   Drum."Step".Ons_StrobeWorkDone := FALSE;
   Drum."Step".Ons_StrobeRejectByCycleInterruption := FALSE;
   Drum."Step".StrobeWorkDone := FALSE;
   Drum."Step".StrobeRejectByCycleInterruption := FALSE;
   Drum."Step".ScSeqOk := FALSE;
   Drum."Step".SeqActive := FALSE;
   Drum.Drive.AlmOk := FALSE;
   Drum.Drive.AlmEmerg := FALSE;
   Drum.Drive.AlmNode := FALSE;
   Drum.Drive.InitPosDrive := FALSE;
   Drum.Drive.InitPosDrivePLS := FALSE;
   Drum.Drive.GearingON := FALSE;
   Drum.Drive.CamHook := FALSE;
   Drum.Drive.CamStoppingPhase := FALSE;
   Drum.Drive.RepositioningRequest := FALSE;
   Drum.Drive.CamRequestResult := FALSE;
   Drum.Drive.CamRequestError := FALSE;
   Drum.Drive.CamRequestOk := TRUE;
   Drum.Drive.CalibDisAxisReq := FALSE;
   Drum.Drive.CalibReq := FALSE;
   Drum.Drive.CalibProcess := FALSE;
   Drum.Drive.HwOvertravelDisReq := FALSE;
   Drum.Drive.HwOvertravelEnReq := FALSE;
   Drum.Drive.AuxCamRequest := FALSE;
   Drum.Drive.TorquePeakEna := FALSE;
   Drum.Drive.Cmd_Repos := FALSE;
   Drum.Drive.Ons_CamRequest := FALSE;
   Drum.Drive.AuxCmdPosition := 0;
   Drum.Drive.Unwind := 90.0;
   Drum.Drive.MaxDev := 30.0;
   Drum.Drive.ReposSpeed := 10.0;
   Drum.Drive.CalcSlaveDifferenceABS := 0.0;
   Drum.Drive.CalcModPosition := 0.0;
   Drum.Drive.CalcSlaveDifference := 0.0;
   Drum.Drive.CalcMinDeltaPos := 0.0;
   Drum.Drive.CalcMaxDeltaPos := 0.0;
   Drum.Drive.CalcHalfPosUnwind := 0.0;
   Drum.Drive.Man.Cmd_PosJog := FALSE;
   Drum.Drive.Man.Cmd_NegJog := FALSE;
   Drum.Drive.Man.Cmd_Step := FALSE;
   Drum.Drive.Man.Cmd_Forward := FALSE;
   Drum.Drive.Man.Cmd_Backward := FALSE;
   Drum.Drive.Man.Cmd_Up := FALSE;
   Drum.Drive.Man.Cmd_Down := FALSE;
   Drum.Drive.Man.Cmd_Intermediate := FALSE;
   Drum.Drive.Man.Cmd_Open := FALSE;
   Drum.Drive.Man.Cmd_Close := FALSE;
   Drum.Drive.Man.Cmd_PreOpen := FALSE;
   Drum.Drive.Man.Cmd_Maintenance := FALSE;
   Drum.Drive.Man.Cmd_OperatorSide := FALSE;
   Drum.Drive.Man.Cmd_NotOperatorSide := FALSE;
   Drum.Drive.Man.Cmd_OnMould := FALSE;
   Drum.Drive.Man.Cmd_OffMould := FALSE;
   Drum.Drive.Man.Cmd_Pos0 := FALSE;
   Drum.Drive.Man.Cmd_Pos1 := FALSE;
   Drum.Drive.Man.Cmd_Pos2 := FALSE;
   Drum.Drive.Man.Cmd_Pos3 := FALSE;
   Drum.Drive.Man.Cmd_Pos4 := FALSE;
   Drum.Drive.Man.Cmd_Pos5 := FALSE;
   Drum.Drive.Man.Ons_Step := FALSE;
   Drum.Drive.Man.PhaseJogCmd := TRUE;
   Drum.Drive.Man.CmdStartStep := FALSE;
   Drum.Drive.Man.CmdEndStep := FALSE;
   Drum.Drive.Man.StepCond := FALSE;
   Drum.Drive.Man.TON_DelayHomeCmd.PT := T#3S;
   Drum.Drive.Man.TON_DelayHomeCmd.IN := FALSE;
   Drum.Drive.Auto.Cmd_Step := FALSE;
   Drum.Drive.Auto.Cmd_StartStep := FALSE;
   Drum.Drive.Auto.Cmd_EndStep := FALSE;
   Drum.Drive.Auto.Cmd_Forward := FALSE;
   Drum.Drive.Auto.Cmd_Backward := FALSE;
   Drum.Drive.Auto.Cmd_Up := FALSE;
   Drum.Drive.Auto.Cmd_Down := FALSE;
   Drum.Drive.Auto.Cmd_Intermediate := FALSE;
   Drum.Drive.Auto.Cmd_Open := FALSE;
   Drum.Drive.Auto.Cmd_Close := FALSE;
   Drum.Drive.Auto.Cmd_PreOpen := FALSE;
   Drum.Drive.Auto.Cmd_Maintenance := FALSE;
   Drum.Drive.Auto.Cmd_OperatorSide := FALSE;
   Drum.Drive.Auto.Cmd_NotOperatorSide := FALSE;
   Drum.Drive.Auto.Cmd_OnMould := FALSE;
   Drum.Drive.Auto.Cmd_OffMould := FALSE;
   Drum.Drive.Auto.Cmd_Pos0 := FALSE;
   Drum.Drive.Auto.Cmd_Pos1 := FALSE;
   Drum.Drive.Auto.Cmd_Pos2 := FALSE;
   Drum.Drive.Auto.Cmd_Pos3 := FALSE;
   Drum.Drive.Auto.Cmd_Pos4 := FALSE;
   Drum.Drive.Auto.Cmd_Pos5 := FALSE;
   Drum.Drive.Auto.Cmd_Gear := FALSE;
   Drum.Drive.ACT.CMD.Enable := FALSE;
   Drum.Drive.ACT.CMD.Pos_Mode := FALSE;
   Drum.Drive.ACT.CMD.MergeDisabled := FALSE;
   Drum.Drive.ACT.CMD.SCurve := FALSE;
   Drum.Drive.ACT.CMD.Cam_Mode := FALSE;
   Drum.Drive.ACT.CMD.Cam_Request := FALSE;
   Drum.Drive.ACT.CMD.Cam_PhaseStop := FALSE;
   Drum.Drive.ACT.CMD.Gear_Mode := FALSE;
   Drum.Drive.ACT.CMD.Repos_Req := FALSE;
   Drum.Drive.ACT.CMD.Jog_Pos := FALSE;
   Drum.Drive.ACT.CMD.Jog_Neg := FALSE;
   Drum.Drive.ACT.CMD.Stop := TRUE;
   Drum.Drive.ACT.CMD.Calibration_Req := FALSE;
   Drum.Drive.ACT.CMD.Reset := FALSE;
   Drum.Drive.ACT.CMD.RegInput1 := FALSE;
   Drum.Drive.ACT.CMD.Brake_Release := FALSE;
   Drum.Drive.ACT.CMD.HwPosOvertravel_Dis := FALSE;
   Drum.Drive.ACT.CMD.HwNegOvertravel_Dis := FALSE;
   Drum.Drive.ACT.CMD.HwOvertravel_MSG_En := FALSE;
   Drum.Drive.ACT.CMD.OneShootMove := FALSE;
   Drum.Drive.ACT.CMD.Move_Type := 3;
   Drum.Drive.ACT.CMD.Target_Pos := 0.0;
   Drum.Drive.ACT.CMD.Speed := 22.0;
   Drum.Drive.ACT.CMD.Acceleration := 200.0;
   Drum.Drive.ACT.CMD.Deceleration := 500.0;
   Drum.Drive.ACT.CMD.Torque_Limit := 30.0;
   Drum.Drive.ACT.CMD.Gear_Ratio := 0.0;
   Drum.Drive.ACT.CMD.Mccp_Length := 0;
   Drum.Drive.ACT.CMD.Mccp_StartSlope := 0.0;
   Drum.Drive.ACT.CMD.Mccp_EndSlope := 0.0;
   Drum.Drive.ACT.CMD.Mapc_Direction := 1;
   Drum.Drive.ACT.CMD.Mapc_SlaveScaling := 1.0;
   Drum.Drive.ACT.CMD.Mapc_MasterScaling := 1.0;
   Drum.Drive.ACT.CMD.Mapc_MasterLockPosition := 67.82901;
   Drum.Drive.ACT.CMD.Mapc_CamLockPosition := 0.0;
   Drum.Drive.ACT.CMD.Cam[0..39].leadingValueStart := 0.0;
   Drum.Drive.ACT.CMD.Cam[0..39].leadingValueEnd := 0.0;
   Drum.Drive.ACT.CMD.Cam[0..39].followingValueStart := 0.0;
   Drum.Drive.ACT.CMD.Cam[0..39].followingValueEnd := 0.0;
   Drum.Drive.ACT.CMD.Cam[0..39].geoVeloStart := 0.0;
   Drum.Drive.ACT.CMD.Cam[0..39].geoVeloEnd := 0.0;
   Drum.Drive.ACT.CMD.Cam[0..39].geoAccelStart := 0.0;
   Drum.Drive.ACT.CMD.Cam[0..39].geoAccelEnd := 0.0;
   Drum.Drive.ACT.CMD.Cam[0..39].geoJerkStart := 0.0;
   Drum.Drive.ACT.CMD.Cam[0..39].geoJerkEnd := 0.0;
   Drum.Drive.ACT.CMD.Cam[0..39].inflectionPointParameter := 0.5;
   Drum.Drive.ACT.CMD.Cam[0..39].modVeloTrapezoidParameter := 1.0;
   Drum.Drive.ACT.CMD.Cam[0..39].modSineMaxAccelCaStar := 0.0;
   Drum.Drive.ACT.CMD.Cam[0..39].camProfileType := 0;
   Drum.Drive.ACT.FBK.Ready := TRUE;
   Drum.Drive.ACT.FBK.Calibrated := TRUE;
   Drum.Drive.ACT.FBK.Fault := FALSE;
   Drum.Drive.ACT.FBK.ModuleConnFault := FALSE;
   Drum.Drive.ACT.FBK.In_Position := FALSE;
   Drum.Drive.ACT.FBK.Standstill := TRUE;
   Drum.Drive.ACT.FBK.Enabled := FALSE;
   Drum.Drive.ACT.FBK.BusReadyStatus := FALSE;
   Drum.Drive.ACT.FBK.BrakeReleased := FALSE;
   Drum.Drive.ACT.FBK.HwPosOvertravelDisabled := FALSE;
   Drum.Drive.ACT.FBK.HwNegOvertravelDisabled := FALSE;
   Drum.Drive.ACT.FBK.SafeOffStatus := FALSE;
   Drum.Drive.ACT.FBK.MaxTorqueLimit := FALSE;
   Drum.Drive.ACT.FBK.PosMerge_IP := FALSE;
   Drum.Drive.ACT.FBK.PosMerge_PC := FALSE;
   Drum.Drive.ACT.FBK.Gearing_IP := FALSE;
   Drum.Drive.ACT.FBK.Position := 89.999;
   Drum.Drive.ACT.FBK.Speed := 0.0;
   Drum.Drive.ACT.FBK.Torque := 0.01220703;
   Drum.Drive.ACT.FBK.RegInput1Pos := 0.0;
   Drum.Drive.ACT.FBK.SeqCamErrorCode := 0;
   Drum.Drive.ACT.FBK.SeqCamTargetPosMAM := 73.57474;
   Drum.Drive.ACT.FBK.SeqCamStatus.EndSequence := FALSE;
   Drum.Drive.ACT.FBK.SeqCamStatus.EndSuccess := FALSE;
   Drum.Drive.ACT.FBK.SeqCamStatus.EndError := FALSE;
   Drum.Drive.ACT.FBK.SeqCamStatus.CamHook := FALSE;
   Drum.Drive.ACT.FBK.SeqCamStatus.BothMapc_IP := FALSE;
   Drum.Drive.ACT.FBK.SeqCamStatus.SlaveFwd := FALSE;
   Drum.Drive.ACT.FBK.SeqCamStatus.SlaveBwd := FALSE;
   Drum.Drive.ACT.FBK.SeqCamStatus.SlaveUnwind := FALSE;
   Drum.Drive.ACT.FBK.SeqCamStatus.WaitValidByOpe := FALSE;
   Drum.Drive.ACT.FBK.SeqCamStatus.MapcA_IP := FALSE;
   Drum.Drive.ACT.FBK.SeqCamStatus.MapcB_IP := FALSE;
   Drum.Drive.ACT.FBK.SeqCamStatus.MapcC_IP := FALSE;
   Drum.Drive.ACT.FBK.SeqCamStatus.CamOnce_PC := FALSE;
   Drum.Drive.ACT.FBK.SeqCamStatus.MaxDevError := FALSE;
   Drum.Drive.ACT.FBK.SeqCamStatus.PositionCamLockStatus := FALSE;
   Drum.Drive.ACT.FBK.SeqCamStatus.WaitRestart := FALSE;
   Drum.Drive.ACT.FBK.SeqCamStatus.Bit17 := FALSE;
   Drum.Drive.ACT.FBK.SeqCamStatus.Bit18 := FALSE;
   Drum.Drive.ACT.FBK.SeqCamStatus.Bit19 := FALSE;
   Drum.Drive.ACT.FBK.SeqCamStatus.Bit20 := FALSE;
   Drum.Drive.ACT.FBK.SeqCamStatus.Bit21 := FALSE;
   Drum.Drive.ACT.FBK.SeqCamStatus.Bit22 := FALSE;
   Drum.Drive.ACT.FBK.SeqCamStatus.Bit23 := FALSE;
   Drum.Drive.ACT.FBK.SeqCamStatus.Bit24 := FALSE;
   Drum.Drive.ACT.FBK.SeqCamStatus.Bit25 := FALSE;
   Drum.Drive.ACT.FBK.SeqCamStatus.Bit26 := FALSE;
   Drum.Drive.ACT.FBK.SeqCamStatus.Bit27 := FALSE;
   Drum.Drive.ACT.FBK.SeqCamStatus.Bit28 := FALSE;
   Drum.Drive.ACT.FBK.SeqCamStatus.Bit29 := FALSE;
   Drum.Drive.ACT.FBK.SeqCamStatus.Bit30 := FALSE;
   Drum.Drive.ACT.FBK.SeqCamStatus.Bit31 := FALSE;
   Drum.Drive.ACT.FBK.SeqCamStatus.Bit32 := FALSE;
   Drum.Drive.PLS.FinePosOk.LowLimit := 89.0;
   Drum.Drive.PLS.FinePosOk.HighLimit := 1.0;
   Drum.Drive.PLS.FinePosOk.Ok := TRUE;
   Drum.Drive.PLS.KeepPosOk.LowLimit := 88.0;
   Drum.Drive.PLS.KeepPosOk.HighLimit := 2.0;
   Drum.Drive.PLS.KeepPosOk.Ok := TRUE;
   Drum.Drive.PLS.Up.LowLimit := 0.0;
   Drum.Drive.PLS.Up.HighLimit := 0.0;
   Drum.Drive.PLS.Up.Ok := FALSE;
   Drum.Drive.PLS.Intermediate.LowLimit := 0.0;
   Drum.Drive.PLS.Intermediate.HighLimit := 0.0;
   Drum.Drive.PLS.Intermediate.Ok := FALSE;
   Drum.Drive.PLS.Down.LowLimit := 0.0;
   Drum.Drive.PLS.Down.HighLimit := 0.0;
   Drum.Drive.PLS.Down.Ok := FALSE;
   Drum.Drive.PLS.Forward.LowLimit := 0.0;
   Drum.Drive.PLS.Forward.HighLimit := 0.0;
   Drum.Drive.PLS.Forward.Ok := FALSE;
   Drum.Drive.PLS.Backward.LowLimit := 0.0;
   Drum.Drive.PLS.Backward.HighLimit := 0.0;
   Drum.Drive.PLS.Backward.Ok := FALSE;
   Drum.Drive.PLS.Open.LowLimit := 0.0;
   Drum.Drive.PLS.Open.HighLimit := 0.0;
   Drum.Drive.PLS.Open.Ok := FALSE;
   Drum.Drive.PLS.Close.LowLimit := 0.0;
   Drum.Drive.PLS.Close.HighLimit := 0.0;
   Drum.Drive.PLS.Close.Ok := FALSE;
   Drum.Drive.PLS.PreOpen.LowLimit := 0.0;
   Drum.Drive.PLS.PreOpen.HighLimit := 0.0;
   Drum.Drive.PLS.PreOpen.Ok := FALSE;
   Drum.Drive.PLS.Maintenance.LowLimit := 0.0;
   Drum.Drive.PLS.Maintenance.HighLimit := 0.0;
   Drum.Drive.PLS.Maintenance.Ok := FALSE;
   Drum.Drive.PLS.OperatorSide.LowLimit := 0.0;
   Drum.Drive.PLS.OperatorSide.HighLimit := 0.0;
   Drum.Drive.PLS.OperatorSide.Ok := FALSE;
   Drum.Drive.PLS.NotOperatorSide.LowLimit := 0.0;
   Drum.Drive.PLS.NotOperatorSide.HighLimit := 0.0;
   Drum.Drive.PLS.NotOperatorSide.Ok := FALSE;
   Drum.Drive.PLS.OnMould.LowLimit := 0.0;
   Drum.Drive.PLS.OnMould.HighLimit := 0.0;
   Drum.Drive.PLS.OnMould.Ok := FALSE;
   Drum.Drive.PLS.OffMould.LowLimit := 0.0;
   Drum.Drive.PLS.OffMould.HighLimit := 0.0;
   Drum.Drive.PLS.OffMould.Ok := FALSE;
   Drum.Drive.PLS.Pos0.LowLimit := 0.0;
   Drum.Drive.PLS.Pos0.HighLimit := 0.0;
   Drum.Drive.PLS.Pos0.Ok := FALSE;
   Drum.Drive.PLS.Pos1.LowLimit := 0.0;
   Drum.Drive.PLS.Pos1.HighLimit := 0.0;
   Drum.Drive.PLS.Pos1.Ok := FALSE;
   Drum.Drive.PLS.Pos2.LowLimit := 0.0;
   Drum.Drive.PLS.Pos2.HighLimit := 0.0;
   Drum.Drive.PLS.Pos2.Ok := FALSE;
   Drum.Drive.PLS.Pos3.LowLimit := 0.0;
   Drum.Drive.PLS.Pos3.HighLimit := 0.0;
   Drum.Drive.PLS.Pos3.Ok := FALSE;
   Drum.Drive.PLS.Pos4.LowLimit := 0.0;
   Drum.Drive.PLS.Pos4.HighLimit := 0.0;
   Drum.Drive.PLS.Pos4.Ok := FALSE;
   Drum.Drive.PLS.Pos5.LowLimit := 0.0;
   Drum.Drive.PLS.Pos5.HighLimit := 0.0;
   Drum.Drive.PLS.Pos5.Ok := FALSE;
   Drum.Drive.TON_EnableDrive.PT := T#500MS;
   Drum.Drive.TON_EnableDrive.IN := FALSE;
   Drum.Drive.TON_HwOvertravel_Dis.PT := T#0MS;
   Drum.Drive.TON_HwOvertravel_Dis.IN := FALSE;
   Drum.Drive.TON_HwOvertravel_En.PT := T#0MS;
   Drum.Drive.TON_HwOvertravel_En.IN := FALSE;
   Drum.Drive.TON_TimeoutMovement.PT := T#20S;
   Drum.Drive.TON_TimeoutMovement.IN := FALSE;
   Drum.Man.OnsSincleCycle := FALSE;
   Drum.Man.CmdSingleCycle := FALSE;
   Drum.Man.EnaPbt := FALSE;
   Drum.Man.RstCmd := TRUE;
   Drum.Man.ScreenNumber := 306_020_301;
   Drum.Man.WithinScreenRange := 0;
   Drum.TON_ScOK.PT := T#20S;
   Drum.TON_ScOK.IN := FALSE;
   DrawerHopper.ScOk := TRUE;
   DrawerHopper.CycleOn := FALSE;
   DrawerHopper.Work := FALSE;
   DrawerHopper.OkToStop := TRUE;
   DrawerHopper.AlmOk := TRUE;
   DrawerHopper.ReqWork := FALSE;
   DrawerHopper.AutoCmd_RunInv := FALSE;
   DrawerHopper.LevReqWork := TRUE;
   DrawerHopper.OutChainObstruction := TRUE;
   DrawerHopper.LevelFiltered := 0.0;
   DrawerHopper.Input.BrkInv := TRUE;
   DrawerHopper.Input.OvrMinLev := FALSE;
   DrawerHopper.Input.OvrMaxLev := FALSE;
   DrawerHopper.Input.WrkLev := FALSE;
   DrawerHopper.Input.CnnIns := FALSE;
   DrawerHopper.Input.TrmSen1 := TRUE;
   DrawerHopper.Input.TrmSen2 := TRUE;
   DrawerHopper.Input.LevPrb.EngValue := 0.0;
   DrawerHopper.Input.LevPrb.ScaledValue := 0.0;
   DrawerHopper.Input.Inv.Flt := TRUE;
   DrawerHopper.Input.Inv.Rdy := FALSE;
   DrawerHopper.Input.Inv.AtRef := TRUE;
   DrawerHopper.Input.Inv.ActSpe := 0.0;
   DrawerHopper.Output.ExtCmd := FALSE;
   DrawerHopper.Output.CmdPwr := FALSE;
   DrawerHopper.Output.Inv.Sta := FALSE;
   DrawerHopper.Output.Inv.Sto := TRUE;
   DrawerHopper.Output.Inv.Rst := FALSE;
   DrawerHopper.Output.Inv.Fwd := TRUE;
   DrawerHopper.Output.Inv.Rev := FALSE;
   DrawerHopper.Output.Inv.Spe := 0.0;
   DrawerHopper.Presence.AnalogSensHprLev := FALSE;
   DrawerHopper.Presence.DigitalSensHprLevDig := TRUE;
   DrawerHopper.Man.CmdStart := FALSE;
   DrawerHopper.Man.CmdStop := FALSE;
   DrawerHopper.Man.EnaPbt := FALSE;
   DrawerHopper.Man.RstCmd := TRUE;
   DrawerHopper.Man.ScreenNumber := 306_030_301;
   DrawerHopper.Man.WithinScreenRange := 0;
   DrawerHopper.TOF_DelayReqWork.PT := T#10S;
   DrawerHopper.TOF_DelayReqWork.IN := FALSE;
   DrawerHopper.TOF_DelayRunInvOff.PT := T#30S;
   DrawerHopper.TOF_DelayRunInvOff.ET := T#30S;
   DrawerHopper.TOF_DelayRunInvOff.IN := FALSE;
   DrawerHopper.TOF_DelayLevReqWork.PT := T#30S;
   DrawerHopper.TOF_DelayLevReqWork.IN := TRUE;
   DrawerHopper.TOF_DelayLevReqWork.Q := TRUE;
   DrawerHopper.TON_ScOk.PT := T#20S;
   DrawerHopper.TON_ScOk.IN := FALSE;
   DrawerHopper.TON_InverterFault.PT := T#15S;
   DrawerHopper.TON_InverterFault.IN := FALSE;
   DrawerHopper.TON_DelayAlmExtraMaxLevel.PT := T#15S;
   DrawerHopper.TON_DelayAlmExtraMaxLevel.IN := FALSE;
   DrawerHopper.TON_DelayAlmExtraMinLevel.PT := T#15S;
   DrawerHopper.TON_DelayAlmExtraMinLevel.IN := FALSE;
   DrawerHopper.TON_DelaySignExtraMaxLevel.PT := T#5S;
   DrawerHopper.TON_DelaySignExtraMaxLevel.IN := FALSE;
   DrawerHopper.TON_DelaySignExtraMinLevel.PT := T#5S;
   DrawerHopper.TON_DelaySignExtraMinLevel.IN := FALSE;
   DrawerHopper.TON_DelayHprLevel.PT := T#5S;
   DrawerHopper.TON_DelayHprLevel.IN := FALSE;
   DrawerProductBelt.ScOk := FALSE;
   DrawerProductBelt.CycleOn := FALSE;
   DrawerProductBelt.Work := FALSE;
   DrawerProductBelt.OkToStop := FALSE;
   DrawerProductBelt.AlmOk := TRUE;
   DrawerProductBelt.ReqWork := FALSE;
   DrawerProductBelt.AutoCmd_RunInv := FALSE;
   DrawerProductBelt.LevReqWork := FALSE;
   DrawerProductBelt.OutChainObstruction := FALSE;
   DrawerProductBelt.LevelFiltered := 0.0;
   DrawerProductBelt.Input.BrkInv := FALSE;
   DrawerProductBelt.Input.OvrMinLev := FALSE;
   DrawerProductBelt.Input.OvrMaxLev := FALSE;
   DrawerProductBelt.Input.WrkLev := FALSE;
   DrawerProductBelt.Input.CnnIns := FALSE;
   DrawerProductBelt.Input.TrmSen1 := FALSE;
   DrawerProductBelt.Input.TrmSen2 := FALSE;
   DrawerProductBelt.Input.LevPrb.EngValue := 0.0;
   DrawerProductBelt.Input.LevPrb.ScaledValue := 0.0;
   DrawerProductBelt.Input.Inv.Flt := FALSE;
   DrawerProductBelt.Input.Inv.Rdy := FALSE;
   DrawerProductBelt.Input.Inv.AtRef := FALSE;
   DrawerProductBelt.Input.Inv.ActSpe := 0.0;
   DrawerProductBelt.Output.ExtCmd := FALSE;
   DrawerProductBelt.Output.CmdPwr := FALSE;
   DrawerProductBelt.Output.Inv.Sta := FALSE;
   DrawerProductBelt.Output.Inv.Sto := FALSE;
   DrawerProductBelt.Output.Inv.Rst := FALSE;
   DrawerProductBelt.Output.Inv.Fwd := FALSE;
   DrawerProductBelt.Output.Inv.Rev := FALSE;
   DrawerProductBelt.Output.Inv.Spe := 0.0;
   DrawerProductBelt.Presence.AnalogSensHprLev := FALSE;
   DrawerProductBelt.Presence.DigitalSensHprLevDig := FALSE;
   DrawerProductBelt.Man.CmdStart := FALSE;
   DrawerProductBelt.Man.CmdStop := FALSE;
   DrawerProductBelt.Man.EnaPbt := FALSE;
   DrawerProductBelt.Man.RstCmd := FALSE;
   DrawerProductBelt.Man.ScreenNumber := 306_040_301;
   DrawerProductBelt.Man.WithinScreenRange := 0;
   DrawerProductBelt.TOF_DelayReqWork.PT := T#10S;
   DrawerProductBelt.TOF_DelayReqWork.IN := FALSE;
   DrawerProductBelt.TOF_DelayRunInvOff.PT := T#30S;
   DrawerProductBelt.TOF_DelayRunInvOff.IN := FALSE;
   DrawerProductBelt.TOF_DelayLevReqWork.PT := T#0MS;
   DrawerProductBelt.TOF_DelayLevReqWork.IN := FALSE;
   DrawerProductBelt.TON_ScOk.PT := T#20S;
   DrawerProductBelt.TON_ScOk.IN := FALSE;
   DrawerProductBelt.TON_InverterFault.PT := T#15S;
   DrawerProductBelt.TON_InverterFault.IN := FALSE;
   DrawerProductBelt.TON_DelayAlmExtraMaxLevel.PT := T#0MS;
   DrawerProductBelt.TON_DelayAlmExtraMaxLevel.IN := FALSE;
   DrawerProductBelt.TON_DelayAlmExtraMinLevel.PT := T#0MS;
   DrawerProductBelt.TON_DelayAlmExtraMinLevel.IN := FALSE;
   DrawerProductBelt.TON_DelaySignExtraMaxLevel.PT := T#0MS;
   DrawerProductBelt.TON_DelaySignExtraMaxLevel.IN := FALSE;
   DrawerProductBelt.TON_DelaySignExtraMinLevel.PT := T#0MS;
   DrawerProductBelt.TON_DelaySignExtraMinLevel.IN := FALSE;
   DrawerProductBelt.TON_DelayHprLevel.PT := T#0MS;
   DrawerProductBelt.TON_DelayHprLevel.IN := FALSE;
   DrawerProductTank.ScOk := FALSE;
   DrawerProductTank.CycleOn := FALSE;
   DrawerProductTank.Work := FALSE;
   DrawerProductTank.OkToStop := FALSE;
   DrawerProductTank.AlmOk := TRUE;
   DrawerProductTank.ReqWork := FALSE;
   DrawerProductTank.AutoCmd_RunInv := FALSE;
   DrawerProductTank.LevReqWork := FALSE;
   DrawerProductTank.OutChainObstruction := FALSE;
   DrawerProductTank.LevelFiltered := 0.0;
   DrawerProductTank.Input.BrkInv := FALSE;
   DrawerProductTank.Input.OvrMinLev := FALSE;
   DrawerProductTank.Input.OvrMaxLev := FALSE;
   DrawerProductTank.Input.WrkLev := FALSE;
   DrawerProductTank.Input.CnnIns := FALSE;
   DrawerProductTank.Input.TrmSen1 := FALSE;
   DrawerProductTank.Input.TrmSen2 := FALSE;
   DrawerProductTank.Input.LevPrb.EngValue := 0.0;
   DrawerProductTank.Input.LevPrb.ScaledValue := 0.0;
   DrawerProductTank.Input.Inv.Flt := FALSE;
   DrawerProductTank.Input.Inv.Rdy := FALSE;
   DrawerProductTank.Input.Inv.AtRef := FALSE;
   DrawerProductTank.Input.Inv.ActSpe := 0.0;
   DrawerProductTank.Output.ExtCmd := FALSE;
   DrawerProductTank.Output.CmdPwr := FALSE;
   DrawerProductTank.Output.Inv.Sta := FALSE;
   DrawerProductTank.Output.Inv.Sto := FALSE;
   DrawerProductTank.Output.Inv.Rst := FALSE;
   DrawerProductTank.Output.Inv.Fwd := FALSE;
   DrawerProductTank.Output.Inv.Rev := FALSE;
   DrawerProductTank.Output.Inv.Spe := 0.0;
   DrawerProductTank.Presence.AnalogSensHprLev := FALSE;
   DrawerProductTank.Presence.DigitalSensHprLevDig := FALSE;
   DrawerProductTank.Man.CmdStart := FALSE;
   DrawerProductTank.Man.CmdStop := FALSE;
   DrawerProductTank.Man.EnaPbt := FALSE;
   DrawerProductTank.Man.RstCmd := FALSE;
   DrawerProductTank.Man.ScreenNumber := 306_050_301;
   DrawerProductTank.Man.WithinScreenRange := 0;
   DrawerProductTank.TOF_DelayReqWork.PT := T#10S;
   DrawerProductTank.TOF_DelayReqWork.IN := FALSE;
   DrawerProductTank.TOF_DelayRunInvOff.PT := T#30S;
   DrawerProductTank.TOF_DelayRunInvOff.IN := FALSE;
   DrawerProductTank.TOF_DelayLevReqWork.PT := T#30S;
   DrawerProductTank.TOF_DelayLevReqWork.IN := FALSE;
   DrawerProductTank.TON_ScOk.PT := T#20S;
   DrawerProductTank.TON_ScOk.IN := FALSE;
   DrawerProductTank.TON_InverterFault.PT := T#15S;
   DrawerProductTank.TON_InverterFault.IN := FALSE;
   DrawerProductTank.TON_DelayAlmExtraMaxLevel.PT := T#15S;
   DrawerProductTank.TON_DelayAlmExtraMaxLevel.IN := FALSE;
   DrawerProductTank.TON_DelayAlmExtraMinLevel.PT := T#15S;
   DrawerProductTank.TON_DelayAlmExtraMinLevel.IN := FALSE;
   DrawerProductTank.TON_DelaySignExtraMaxLevel.PT := T#5S;
   DrawerProductTank.TON_DelaySignExtraMaxLevel.IN := FALSE;
   DrawerProductTank.TON_DelaySignExtraMinLevel.PT := T#5S;
   DrawerProductTank.TON_DelaySignExtraMinLevel.IN := FALSE;
   DrawerProductTank.TON_DelayHprLevel.PT := T#5S;
   DrawerProductTank.TON_DelayHprLevel.IN := FALSE;
   DrumBrush.ScOk := TRUE;
   DrumBrush.CycleOn := FALSE;
   DrumBrush.Work := FALSE;
   DrumBrush.OkToStop := TRUE;
   DrumBrush.AlmOk := TRUE;
   DrumBrush.ReqWork := FALSE;
   DrumBrush.AutoCmd_RunInv := FALSE;
   DrumBrush.LevReqWork := TRUE;
   DrumBrush.OutChainObstruction := TRUE;
   DrumBrush.LevelFiltered := 0.0;
   DrumBrush.Input.BrkInv := FALSE;
   DrumBrush.Input.OvrMinLev := FALSE;
   DrumBrush.Input.OvrMaxLev := FALSE;
   DrumBrush.Input.WrkLev := FALSE;
   DrumBrush.Input.CnnIns := FALSE;
   DrumBrush.Input.TrmSen1 := FALSE;
   DrumBrush.Input.TrmSen2 := FALSE;
   DrumBrush.Input.LevPrb.EngValue := 0.0;
   DrumBrush.Input.LevPrb.ScaledValue := 0.0;
   DrumBrush.Input.Inv.Flt := FALSE;
   DrumBrush.Input.Inv.Rdy := FALSE;
   DrumBrush.Input.Inv.AtRef := FALSE;
   DrumBrush.Input.Inv.ActSpe := 0.0;
   DrumBrush.Output.ExtCmd := TRUE;
   DrumBrush.Output.CmdPwr := FALSE;
   DrumBrush.Output.Inv.Sta := FALSE;
   DrumBrush.Output.Inv.Sto := TRUE;
   DrumBrush.Output.Inv.Rst := FALSE;
   DrumBrush.Output.Inv.Fwd := TRUE;
   DrumBrush.Output.Inv.Rev := FALSE;
   DrumBrush.Output.Inv.Spe := 35.0;
   DrumBrush.Presence.AnalogSensHprLev := FALSE;
   DrumBrush.Presence.DigitalSensHprLevDig := FALSE;
   DrumBrush.Man.CmdStart := FALSE;
   DrumBrush.Man.CmdStop := FALSE;
   DrumBrush.Man.EnaPbt := FALSE;
   DrumBrush.Man.RstCmd := TRUE;
   DrumBrush.Man.ScreenNumber := 306_060_301;
   DrumBrush.Man.WithinScreenRange := 0;
   DrumBrush.TOF_DelayReqWork.PT := T#10S;
   DrumBrush.TOF_DelayReqWork.IN := FALSE;
   DrumBrush.TOF_DelayRunInvOff.PT := T#30S;
   DrumBrush.TOF_DelayRunInvOff.IN := FALSE;
   DrumBrush.TOF_DelayLevReqWork.PT := T#30S;
   DrumBrush.TOF_DelayLevReqWork.IN := TRUE;
   DrumBrush.TON_ScOk.PT := T#20S;
   DrumBrush.TON_ScOk.IN := FALSE;
   DrumBrush.TON_InverterFault.PT := T#15S;
   DrumBrush.TON_InverterFault.IN := FALSE;
   DrumBrush.TON_DelayAlmExtraMaxLevel.PT := T#15S;
   DrumBrush.TON_DelayAlmExtraMaxLevel.IN := FALSE;
   DrumBrush.TON_DelayAlmExtraMinLevel.PT := T#15S;
   DrumBrush.TON_DelayAlmExtraMinLevel.IN := FALSE;
   DrumBrush.TON_DelaySignExtraMaxLevel.PT := T#5S;
   DrumBrush.TON_DelaySignExtraMaxLevel.IN := FALSE;
   DrumBrush.TON_DelaySignExtraMinLevel.PT := T#5S;
   DrumBrush.TON_DelaySignExtraMinLevel.IN := FALSE;
   DrumBrush.TON_DelayHprLevel.PT := T#5S;
   DrumBrush.TON_DelayHprLevel.IN := FALSE;
   DrumProductBelt.ScOk := TRUE;
   DrumProductBelt.CycleOn := FALSE;
   DrumProductBelt.Work := FALSE;
   DrumProductBelt.OkToStop := TRUE;
   DrumProductBelt.AlmOk := TRUE;
   DrumProductBelt.ReqWork := TRUE;
   DrumProductBelt.AutoCmd_RunInv := FALSE;
   DrumProductBelt.LevReqWork := FALSE;
   DrumProductBelt.OutChainObstruction := TRUE;
   DrumProductBelt.LevelFiltered := 0.0;
   DrumProductBelt.Input.BrkInv := FALSE;
   DrumProductBelt.Input.OvrMinLev := FALSE;
   DrumProductBelt.Input.OvrMaxLev := FALSE;
   DrumProductBelt.Input.WrkLev := FALSE;
   DrumProductBelt.Input.CnnIns := FALSE;
   DrumProductBelt.Input.TrmSen1 := TRUE;
   DrumProductBelt.Input.TrmSen2 := TRUE;
   DrumProductBelt.Input.LevPrb.EngValue := 0.0;
   DrumProductBelt.Input.LevPrb.ScaledValue := 0.0;
   DrumProductBelt.Input.Inv.Flt := FALSE;
   DrumProductBelt.Input.Inv.Rdy := FALSE;
   DrumProductBelt.Input.Inv.AtRef := FALSE;
   DrumProductBelt.Input.Inv.ActSpe := 0.0;
   DrumProductBelt.Output.ExtCmd := FALSE;
   DrumProductBelt.Output.CmdPwr := FALSE;
   DrumProductBelt.Output.Inv.Sta := FALSE;
   DrumProductBelt.Output.Inv.Sto := TRUE;
   DrumProductBelt.Output.Inv.Rst := FALSE;
   DrumProductBelt.Output.Inv.Fwd := TRUE;
   DrumProductBelt.Output.Inv.Rev := FALSE;
   DrumProductBelt.Output.Inv.Spe := 70.0;
   DrumProductBelt.Presence.AnalogSensHprLev := FALSE;
   DrumProductBelt.Presence.DigitalSensHprLevDig := FALSE;
   DrumProductBelt.Man.CmdStart := FALSE;
   DrumProductBelt.Man.CmdStop := FALSE;
   DrumProductBelt.Man.EnaPbt := FALSE;
   DrumProductBelt.Man.RstCmd := TRUE;
   DrumProductBelt.Man.ScreenNumber := 306_070_301;
   DrumProductBelt.Man.WithinScreenRange := 0;
   DrumProductBelt.TOF_DelayReqWork.PT := T#10S;
   DrumProductBelt.TOF_DelayReqWork.IN := TRUE;
   DrumProductBelt.TOF_DelayRunInvOff.PT := T#10S;
   DrumProductBelt.TOF_DelayRunInvOff.IN := FALSE;
   DrumProductBelt.TOF_DelayLevReqWork.PT := T#0MS;
   DrumProductBelt.TOF_DelayLevReqWork.IN := FALSE;
   DrumProductBelt.TON_ScOk.PT := T#20S;
   DrumProductBelt.TON_ScOk.IN := FALSE;
   DrumProductBelt.TON_InverterFault.PT := T#15S;
   DrumProductBelt.TON_InverterFault.IN := FALSE;
   DrumProductBelt.TON_DelayAlmExtraMaxLevel.PT := T#0MS;
   DrumProductBelt.TON_DelayAlmExtraMaxLevel.IN := FALSE;
   DrumProductBelt.TON_DelayAlmExtraMinLevel.PT := T#0MS;
   DrumProductBelt.TON_DelayAlmExtraMinLevel.IN := FALSE;
   DrumProductBelt.TON_DelaySignExtraMaxLevel.PT := T#0MS;
   DrumProductBelt.TON_DelaySignExtraMaxLevel.IN := FALSE;
   DrumProductBelt.TON_DelaySignExtraMinLevel.PT := T#0MS;
   DrumProductBelt.TON_DelaySignExtraMinLevel.IN := FALSE;
   DrumProductBelt.TON_DelayHprLevel.PT := T#0MS;
   DrumProductBelt.TON_DelayHprLevel.IN := FALSE;
   DrumProductTank.ScOk := TRUE;
   DrumProductTank.CycleOn := FALSE;
   DrumProductTank.Work := FALSE;
   DrumProductTank.OkToStop := TRUE;
   DrumProductTank.AlmOk := TRUE;
   DrumProductTank.ReqWork := TRUE;
   DrumProductTank.AutoCmd_RunInv := FALSE;
   DrumProductTank.LevReqWork := FALSE;
   DrumProductTank.OutChainObstruction := TRUE;
   DrumProductTank.LevelFiltered := 0.0;
   DrumProductTank.Input.BrkInv := FALSE;
   DrumProductTank.Input.OvrMinLev := FALSE;
   DrumProductTank.Input.OvrMaxLev := FALSE;
   DrumProductTank.Input.WrkLev := FALSE;
   DrumProductTank.Input.CnnIns := FALSE;
   DrumProductTank.Input.TrmSen1 := FALSE;
   DrumProductTank.Input.TrmSen2 := FALSE;
   DrumProductTank.Input.LevPrb.EngValue := 0.0;
   DrumProductTank.Input.LevPrb.ScaledValue := 0.0;
   DrumProductTank.Input.Inv.Flt := FALSE;
   DrumProductTank.Input.Inv.Rdy := FALSE;
   DrumProductTank.Input.Inv.AtRef := FALSE;
   DrumProductTank.Input.Inv.ActSpe := 0.0;
   DrumProductTank.Output.ExtCmd := FALSE;
   DrumProductTank.Output.CmdPwr := FALSE;
   DrumProductTank.Output.Inv.Sta := FALSE;
   DrumProductTank.Output.Inv.Sto := TRUE;
   DrumProductTank.Output.Inv.Rst := FALSE;
   DrumProductTank.Output.Inv.Fwd := TRUE;
   DrumProductTank.Output.Inv.Rev := FALSE;
   DrumProductTank.Output.Inv.Spe := 35.0;
   DrumProductTank.Presence.AnalogSensHprLev := FALSE;
   DrumProductTank.Presence.DigitalSensHprLevDig := FALSE;
   DrumProductTank.Man.CmdStart := FALSE;
   DrumProductTank.Man.CmdStop := FALSE;
   DrumProductTank.Man.EnaPbt := FALSE;
   DrumProductTank.Man.RstCmd := TRUE;
   DrumProductTank.Man.ScreenNumber := 306_080_301;
   DrumProductTank.Man.WithinScreenRange := 0;
   DrumProductTank.TOF_DelayReqWork.PT := T#10S;
   DrumProductTank.TOF_DelayReqWork.IN := TRUE;
   DrumProductTank.TOF_DelayRunInvOff.PT := T#30S;
   DrumProductTank.TOF_DelayRunInvOff.IN := FALSE;
   DrumProductTank.TOF_DelayLevReqWork.PT := T#30S;
   DrumProductTank.TOF_DelayLevReqWork.IN := FALSE;
   DrumProductTank.TON_ScOk.PT := T#20S;
   DrumProductTank.TON_ScOk.IN := FALSE;
   DrumProductTank.TON_InverterFault.PT := T#15S;
   DrumProductTank.TON_InverterFault.IN := FALSE;
   DrumProductTank.TON_DelayAlmExtraMaxLevel.PT := T#15S;
   DrumProductTank.TON_DelayAlmExtraMaxLevel.IN := FALSE;
   DrumProductTank.TON_DelayAlmExtraMinLevel.PT := T#15S;
   DrumProductTank.TON_DelayAlmExtraMinLevel.IN := FALSE;
   DrumProductTank.TON_DelaySignExtraMaxLevel.PT := T#5S;
   DrumProductTank.TON_DelaySignExtraMaxLevel.IN := FALSE;
   DrumProductTank.TON_DelaySignExtraMinLevel.PT := T#5S;
   DrumProductTank.TON_DelaySignExtraMinLevel.IN := FALSE;
   DrumProductTank.TON_DelayHprLevel.PT := T#5S;
   DrumProductTank.TON_DelayHprLevel.IN := FALSE;
   HorizontalVib.Cfg_0_Drive_1_Pneum := FALSE;
   HorizontalVib.Cfg_CmdMouldBlock := FALSE;
   HorizontalVib.Presence_Sensors := FALSE;
   HorizontalVib.ScOk := FALSE;
   HorizontalVib.CycleOn := FALSE;
   HorizontalVib.Work := FALSE;
   HorizontalVib.OkToStop := FALSE;
   HorizontalVib.AlmOk := FALSE;
   HorizontalVib.OutChainObstruction := FALSE;
   HorizontalVib.Ons_TimeWork := FALSE;
   HorizontalVib.Ons_StrobeWork := FALSE;
   HorizontalVib.Ons_WorkReqPosition := FALSE;
   HorizontalVib.SingleCycle := FALSE;
   HorizontalVib.WorkReqPosition := 0.0;
   HorizontalVib.Input.EnaSel := FALSE;
   HorizontalVib.Input.MouBlk1On := FALSE;
   HorizontalVib.Input.MouBlk1Off := FALSE;
   HorizontalVib.Input.MouBlk2On := FALSE;
   HorizontalVib.Input.MouBlk2Off := FALSE;
   HorizontalVib.Output.EnaSelLgh := FALSE;
   HorizontalVib.Output.CmdMouBlk1On := FALSE;
   HorizontalVib.Output.CmdMouBlk1Off := FALSE;
   HorizontalVib.Output.CmdMouBlk2On := FALSE;
   HorizontalVib.Output.CmdMouBlk2Off := FALSE;
   HorizontalVib.Drive.AutoCmd_RunInv := FALSE;
   HorizontalVib.Drive.Input.BrkInv := FALSE;
   HorizontalVib.Drive.Input.BrkMot1 := FALSE;
   HorizontalVib.Drive.Input.BrkMot2 := FALSE;
   HorizontalVib.Drive.Input.TrmSen1 := FALSE;
   HorizontalVib.Drive.Input.TrmSen2 := FALSE;
   HorizontalVib.Drive.Input.Inv.Flt := FALSE;
   HorizontalVib.Drive.Input.Inv.Rdy := FALSE;
   HorizontalVib.Drive.Input.Inv.AtRef := FALSE;
   HorizontalVib.Drive.Input.Inv.ActSpe := 0.0;
   HorizontalVib.Drive.Output.CmdPwr := FALSE;
   HorizontalVib.Drive.Output.Inv.Sta := FALSE;
   HorizontalVib.Drive.Output.Inv.Sto := FALSE;
   HorizontalVib.Drive.Output.Inv.Rst := FALSE;
   HorizontalVib.Drive.Output.Inv.Fwd := FALSE;
   HorizontalVib.Drive.Output.Inv.Rev := FALSE;
   HorizontalVib.Drive.Output.Inv.Spe := 0.0;
   HorizontalVib.Drive.Man.CmdStart := FALSE;
   HorizontalVib.Drive.Man.CmdStop := FALSE;
   HorizontalVib.Drive.TOF_DelayRunInvOff.PT := T#0MS;
   HorizontalVib.Drive.TOF_DelayRunInvOff.IN := FALSE;
   HorizontalVib.Drive.TON_InverterFault.PT := T#0MS;
   HorizontalVib.Drive.TON_InverterFault.IN := FALSE;
   HorizontalVib.Man.CmdMouBlk1On := FALSE;
   HorizontalVib.Man.CmdMouBlk1Off := FALSE;
   HorizontalVib.Man.CmdMouBlk2On := FALSE;
   HorizontalVib.Man.CmdMouBlk2Off := FALSE;
   HorizontalVib.Man.Ons_SingleCycle := FALSE;
   HorizontalVib.Man.CmdSingleCycle := FALSE;
   HorizontalVib.Man.EnaPbt := FALSE;
   HorizontalVib.Man.RstCmd := FALSE;
   HorizontalVib.Man.ScreenNumber := 306_090_301;
   HorizontalVib.Man.WithinScreenRange := 0;
   HorizontalVib.Pneum.Input.LowPos := FALSE;
   HorizontalVib.Pneum.Input.HigPos := FALSE;
   HorizontalVib.Pneum.Input.AirPrsExtOk := FALSE;
   HorizontalVib.Pneum.Input.AirPrsIntOk := FALSE;
   HorizontalVib.Pneum.Input.FbkPrsExt.EngValue := 0.0;
   HorizontalVib.Pneum.Input.FbkPrsExt.ScaledValue := 0.0;
   HorizontalVib.Pneum.Input.FbkPrsInt.EngValue := 0.0;
   HorizontalVib.Pneum.Input.FbkPrsInt.ScaledValue := 0.0;
   HorizontalVib.Pneum.Output.LowPos := FALSE;
   HorizontalVib.Pneum.Output.HigPos := FALSE;
   HorizontalVib.Pneum.Output.CmdVib := FALSE;
   HorizontalVib.Pneum.Output.CmdLowPrs := FALSE;
   HorizontalVib.Pneum.Output.CmdPrsExt.EngValue := 0.0;
   HorizontalVib.Pneum.Output.CmdPrsExt.ScaledValue := 0.0;
   HorizontalVib.Pneum.Output.CmdPrsInt.EngValue := 0.0;
   HorizontalVib.Pneum.Output.CmdPrsInt.ScaledValue := 0.0;
   HorizontalVib.Pneum.Presence.PressSwitchExt := FALSE;
   HorizontalVib.Pneum.Presence.PressSwitchInt := FALSE;
   HorizontalVib.Pneum.Presence.Riser := FALSE;
   HorizontalVib.Pneum.Man.CmdVibOn := FALSE;
   HorizontalVib.Pneum.Man.CmdVibOff := FALSE;
   HorizontalVib.Pneum.Man.CmdVibUp := FALSE;
   HorizontalVib.Pneum.Man.CmdVibDown := FALSE;
   HorizontalVib.Pneum.TON_AlmPosVib.PT := T#0MS;
   HorizontalVib.Pneum.TON_AlmPosVib.IN := FALSE;
   HorizontalVib.Pneum.TON_AlmPrsExt.PT := T#0MS;
   HorizontalVib.Pneum.TON_AlmPrsExt.IN := FALSE;
   HorizontalVib.Pneum.TON_AlmPrsInt.PT := T#0MS;
   HorizontalVib.Pneum.TON_AlmPrsInt.IN := FALSE;
   HorizontalVib."Step"._00_CycleActivated := FALSE;
   HorizontalVib."Step"._05_MouBlkOnCmd := FALSE;
   HorizontalVib."Step"._10_MouBlkOnPos_VibrationTime := FALSE;
   HorizontalVib."Step"._20_WorkDone_VibOffCmd := FALSE;
   HorizontalVib."Step"._30_VibOff_MouBlkOffCmd := FALSE;
   HorizontalVib."Step"._40_MouBlkOffPos_CycleEnd := FALSE;
   HorizontalVib."Step".Ons_StrobeWorkDone := FALSE;
   HorizontalVib."Step".StrobeWorkDone := FALSE;
   HorizontalVib."Step".ScSeqOk := FALSE;
   HorizontalVib."Step".SeqActive := FALSE;
   HorizontalVib."Step".TON_VibMouBlk1On.PT := T#0MS;
   HorizontalVib."Step".TON_VibMouBlk1On.IN := FALSE;
   HorizontalVib."Step".TON_VibMouBlk2On.PT := T#0MS;
   HorizontalVib."Step".TON_VibMouBlk2On.IN := FALSE;
   HorizontalVib."Step".TON_WaitingMouBlkOn.PT := T#0MS;
   HorizontalVib."Step".TON_WaitingMouBlkOn.IN := FALSE;
   HorizontalVib."Step".TON_WaitingMouBlkOff.PT := T#0MS;
   HorizontalVib."Step".TON_WaitingMouBlkOff.IN := FALSE;
   HorizontalVib."Step".TON_WaitingVibOff.PT := T#0MS;
   HorizontalVib."Step".TON_WaitingVibOff.IN := FALSE;
   HorizontalVib."Step".TON_TimeVibration.PT := T#0MS;
   HorizontalVib."Step".TON_TimeVibration.IN := FALSE;
   HorizontalVib.RTO_Work.PT := T#0MS;
   HorizontalVib.RTO_Work.IN := FALSE;
   HorizontalVib.TON_ScOk.PT := T#0MS;
   HorizontalVib.TON_ScOk.IN := FALSE;
   HorizontalVib.TON_TimeoutWork.PT := T#0MS;
   HorizontalVib.TON_TimeoutWork.IN := FALSE;
   HorizontalVib.TON_AlmMouldBlock1.PT := T#0MS;
   HorizontalVib.TON_AlmMouldBlock1.IN := FALSE;
   HorizontalVib.TON_AlmMouldBlock2.PT := T#0MS;
   HorizontalVib.TON_AlmMouldBlock2.IN := FALSE;
END_DATA_BLOCK
